PROGRAM AXIS_1
VAR
END_VAR

//Initial parameters of an Axis
(*IF _TaskInfo[fbGetCurTaskIndex.index].FirstCycle THEN
    //Axis description for EPICS PV
    GVL.astAxes[1].stDescription.sAxisName := 'MotorApplication1';
    GVL.astAxes[1].stDescription.eUnit := E_AxisEngUnit.eMeter;
    GVL.astAxes[1].stDescription.nPrefix := -3;

    //Initial default values:
    GVL.astAxes[1].stConfig.eHomeSeq := 0;
    GVL.astAxes[1].stConfig.fHomePosition := 0.0;
    GVL.astAxes[1].stConfig.fHomeFinishDistance := 0.0;
    GVL.astAxes[1].stConfig.eRestorePosition := E_RestorePosition.eRestoreWithoutHome;
	
END_IF*)

(*Simons Idea of linking axis to outputs
stSafetyData.aSafetyOuputs[1].abLinkedAxes[1] := TRUE;
stSafetyData.aSafetyOuputs[2].abLinkedAxes[1] := TRUE;
stSafetyData.aSafetyOuputs[3].abLinkedAxes[1] := TRUE;
stSafetyData.aSafetyOuputs[4].abLinkedAxes[1] := TRUE;
stSafetyData.aSafetyOuputs[5].abLinkedAxes[1] := TRUE;
stSafetyData.aSafetyOuputs[6].abLinkedAxes[1] := TRUE;
stSafetyData.aSafetyOuputs[7].abLinkedAxes[1] := TRUE;
stSafetyData.aSafetyOuputs[8].abLinkedAxes[1] := TRUE;
stSafetyData.aSafetyOuputs[9].abLinkedAxes[1] := TRUE;
*)

//Define ACTIONS() or write exclusive code for an specific axis.
(*Eg. Stop when temperature reaches certain values, reduce speed if  a signal is activated, etc.
Eg. GVL.astAxes[x].stControl.bInterlockFwd := NOT bInterlockFwdOK;*)
GVL.astAxes[1].stConfig.eRestorePosition:=1;
GVL.astAxes[1].stSafety.iSafetyOutputGroup := 1; //Sets the group this axis will be in, groups defined in main.group prg

END_PROGRAM

(* stored: Version 1.1.0.1, ProductVersion 3.1.4024.11
   POU AXIS_1: Id {a91ca9eb-6cf6-44ae-b18e-e212bef47c21}, SpecialFunc None *)
